(* IEC 61131-3 sources: festo-codesys-mcp/knowledge/library/actuators, 5 files *)

(* ---- FB_ButtonLamp.st ---- *)
(* =============================================================
   FB_ButtonLamp — Illuminated Pushbutton Controller

   Category:     Actuators
   Platform:     CODESYS V3.5 (IEC 61131-3)
   Version:      1.0
   Dependencies: None (standard IEC only)

   Controls an illuminated pushbutton with multiple lamp modes:
   - OFF: Lamp off
   - ON: Lamp solid on
   - BLINK_SLOW: 1Hz blink (500ms on / 500ms off)
   - BLINK_FAST: 4Hz blink (125ms on / 125ms off)

   Also provides edge detection on the button input.

   Usage:
     fbStart : FB_ButtonLamp;
     fbStart(bButton := bDI_StartBtn, nLampMode := 1);
     bStartPressed := fbStart.bPressed;
     bStartLamp    := fbStart.bLamp;
   ============================================================= *)
FUNCTION_BLOCK FB_ButtonLamp
VAR_INPUT
    bButton     : BOOL;                (* Button input (NO contact) *)
    nLampMode   : INT := 0;            (* 0=OFF, 1=ON, 2=BLINK_SLOW, 3=BLINK_FAST *)
END_VAR
VAR_OUTPUT
    bLamp       : BOOL;                (* Lamp output *)
    bPressed    : BOOL;                (* Button is pressed (debounced) *)
    bRising     : BOOL;                (* Rising edge on button *)
    bFalling    : BOOL;                (* Falling edge on button *)
END_VAR
VAR
    tonDebounce : TON;
    rtrigBtn    : R_TRIG;
    ftrigBtn    : F_TRIG;
    tonBlinkOn  : TON;
    tonBlinkOff : TON;
    bBlinkState : BOOL;
    tOnTime     : TIME;
    tOffTime    : TIME;
END_VAR

(* Debounce button *)
tonDebounce(IN := bButton, PT := T#30MS);
bPressed := tonDebounce.Q;

(* Edge detection *)
rtrigBtn(CLK := bPressed);
ftrigBtn(CLK := bPressed);
bRising := rtrigBtn.Q;
bFalling := ftrigBtn.Q;

(* Lamp control *)
CASE nLampMode OF
0: (* OFF *)
    bLamp := FALSE;

1: (* Solid ON *)
    bLamp := TRUE;

2: (* Blink slow — 1Hz *)
    tOnTime := T#500MS;
    tOffTime := T#500MS;
    IF NOT bBlinkState THEN
        tonBlinkOff(IN := TRUE, PT := tOffTime);
        IF tonBlinkOff.Q THEN
            bBlinkState := TRUE;
            tonBlinkOff(IN := FALSE, PT := tOffTime);
        END_IF
    ELSE
        tonBlinkOn(IN := TRUE, PT := tOnTime);
        IF tonBlinkOn.Q THEN
            bBlinkState := FALSE;
            tonBlinkOn(IN := FALSE, PT := tOnTime);
        END_IF
    END_IF
    bLamp := bBlinkState;

3: (* Blink fast — 4Hz *)
    tOnTime := T#125MS;
    tOffTime := T#125MS;
    IF NOT bBlinkState THEN
        tonBlinkOff(IN := TRUE, PT := tOffTime);
        IF tonBlinkOff.Q THEN
            bBlinkState := TRUE;
            tonBlinkOff(IN := FALSE, PT := tOffTime);
        END_IF
    ELSE
        tonBlinkOn(IN := TRUE, PT := tOnTime);
        IF tonBlinkOn.Q THEN
            bBlinkState := FALSE;
            tonBlinkOn(IN := FALSE, PT := tOnTime);
        END_IF
    END_IF
    bLamp := bBlinkState;

ELSE
    bLamp := FALSE;
END_CASE

END_FUNCTION_BLOCK

(* ---- FB_PneumaticCylinder.st ---- *)
(* =============================================================
   FB_PneumaticCylinder — Pneumatic Cylinder Controller

   Category:     Actuators
   Platform:     CODESYS V3.5 (IEC 61131-3)
   Version:      1.0
   Dependencies: None (standard IEC only)

   Controls single-acting or double-acting pneumatic cylinders
   with optional limit switch feedback and timeout monitoring.

   Features:
   - Extend/retract commands with edge detection
   - Limit switch monitoring (extended/retracted sensors)
   - Configurable timeout for fault detection
   - Manual/auto mode support

   Usage:
     fbClamp : FB_PneumaticCylinder;
     fbClamp(bExtend := bCmdClamp, bRetract := bCmdUnclamp,
             bSnsExtended := bDI_ClampFwd, bSnsRetracted := bDI_ClampRev,
             tTimeout := T#3S);
     bClamped   := fbClamp.bExtended;
     bUnclamped := fbClamp.bRetracted;
     bFault     := fbClamp.bErr;
   ============================================================= *)
FUNCTION_BLOCK FB_PneumaticCylinder
VAR_INPUT
    bExtend         : BOOL;                (* Command: extend cylinder *)
    bRetract        : BOOL;                (* Command: retract cylinder *)
    bSnsExtended    : BOOL;                (* Sensor: fully extended *)
    bSnsRetracted   : BOOL;                (* Sensor: fully retracted *)
    tTimeout        : TIME := T#5S;        (* Motion timeout *)
    bDoubleActing   : BOOL := TRUE;        (* TRUE=double-acting, FALSE=spring-return *)
    bEnable         : BOOL := TRUE;        (* Enable control *)
    bReset          : BOOL;                (* Reset error *)
END_VAR
VAR_OUTPUT
    bSolExtend      : BOOL;                (* Solenoid: extend valve *)
    bSolRetract     : BOOL;                (* Solenoid: retract valve (double-acting only) *)
    bExtended       : BOOL;                (* Status: fully extended *)
    bRetracted      : BOOL;                (* Status: fully retracted *)
    bMoving         : BOOL;                (* Status: in motion *)
    bErr          : BOOL;                (* Error: timeout or sensor conflict *)
    nErrId          : DINT;                 (* 0=OK, 1=Extend timeout, 2=Retract timeout, 3=Sensor conflict *)
END_VAR
VAR
    nState          : INT := 0;            (* 0=Idle, 1=Extending, 2=Extended, 3=Retracting, 4=Retracted, 10=Error *)
    tonTimeout      : TON;
    rtrigExtend     : R_TRIG;
    rtrigRetract    : R_TRIG;
END_VAR

rtrigExtend(CLK := bExtend);
rtrigRetract(CLK := bRetract);

(* Sensor conflict detection *)
IF bSnsExtended AND bSnsRetracted THEN
    nState := 10;
    nErrId := 3;
    bErr := TRUE;
    bSolExtend := FALSE;
    bSolRetract := FALSE;
END_IF

(* Reset *)
IF bReset AND bErr THEN
    nState := 0;
    bErr := FALSE;
    nErrId := 0;
    tonTimeout(IN := FALSE, PT := tTimeout);
END_IF

IF NOT bEnable THEN
    bSolExtend := FALSE;
    bSolRetract := FALSE;
    bMoving := FALSE;
    RETURN;
END_IF

CASE nState OF
0: (* Idle *)
    bSolExtend := FALSE;
    bSolRetract := FALSE;
    bMoving := FALSE;
    bExtended := bSnsExtended;
    bRetracted := bSnsRetracted;

    IF rtrigExtend.Q AND NOT bSnsExtended THEN
        nState := 1;
    ELSIF rtrigRetract.Q AND NOT bSnsRetracted THEN
        nState := 3;
    END_IF

1: (* Extending *)
    bSolExtend := TRUE;
    IF bDoubleActing THEN bSolRetract := FALSE; END_IF
    bMoving := TRUE;
    tonTimeout(IN := TRUE, PT := tTimeout);

    IF bSnsExtended THEN
        nState := 2;
        tonTimeout(IN := FALSE, PT := tTimeout);
    ELSIF tonTimeout.Q THEN
        nState := 10;
        nErrId := 1;
        bErr := TRUE;
        bSolExtend := FALSE;
    END_IF

2: (* Extended — hold position *)
    bSolExtend := TRUE;
    IF bDoubleActing THEN bSolRetract := FALSE; END_IF
    bMoving := FALSE;
    bExtended := TRUE;
    bRetracted := FALSE;

    IF rtrigRetract.Q THEN
        nState := 3;
    END_IF

3: (* Retracting *)
    bSolExtend := FALSE;
    IF bDoubleActing THEN bSolRetract := TRUE; END_IF
    bMoving := TRUE;
    tonTimeout(IN := TRUE, PT := tTimeout);

    IF bSnsRetracted THEN
        nState := 4;
        tonTimeout(IN := FALSE, PT := tTimeout);
    ELSIF tonTimeout.Q THEN
        nState := 10;
        nErrId := 2;
        bErr := TRUE;
        IF bDoubleActing THEN bSolRetract := FALSE; END_IF
    END_IF

4: (* Retracted — hold position *)
    bSolExtend := FALSE;
    IF bDoubleActing THEN bSolRetract := FALSE; END_IF
    bMoving := FALSE;
    bExtended := FALSE;
    bRetracted := TRUE;

    IF rtrigExtend.Q THEN
        nState := 1;
    END_IF

10: (* Error *)
    bSolExtend := FALSE;
    bSolRetract := FALSE;
    bMoving := FALSE;

END_CASE

END_FUNCTION_BLOCK

(* ---- FB_PumpManager.st ---- *)
(* =============================================================
   FB_PumpManager — Dual Pump Coordination with Failover

   Category:     Actuators
   Platform:     CODESYS V3.5 (IEC 61131-3)
   Version:      1.0
   Dependencies: None (standard IEC only)

   Manages two pumps with automatic failover, runtime
   equalization, and maintenance hour tracking. Alternates
   primary pump based on accumulated runtime.

   Usage:
     fbPumps : FB_PumpManager;
     fbPumps(
       bEnable   := bCoolingEnable,
       bFlowOK   := bFlowSwitch,
       bPump1OK  := NOT bPump1Fault,
       bPump2OK  := NOT bPump2Fault
     );
     bPump1 := fbPumps.bPump1;
     bPump2 := fbPumps.bPump2;
   ============================================================= *)
FUNCTION_BLOCK FB_PumpManager
VAR_INPUT
    bEnable             : BOOL;             (* Enable pump system *)
    bFlowOK             : BOOL;             (* Flow sensor feedback *)
    bPump1OK            : BOOL := TRUE;     (* Pump 1 healthy *)
    bPump2OK            : BOOL := TRUE;     (* Pump 2 healthy *)
    bSwapPumps          : BOOL;             (* Manual swap command *)
    tFlowCheckDelay     : TIME := T#5S;     (* Delay before flow check *)
    nHoursToSwap        : DINT := 100;      (* Runtime hours before auto-swap *)
END_VAR
VAR_OUTPUT
    bPump1              : BOOL;             (* Pump 1 output *)
    bPump2              : BOOL;             (* Pump 2 output *)
    bFlowAlarm          : BOOL;             (* No flow detected *)
    bBothFaulted        : BOOL;             (* Both pumps faulted *)
    bPumpActive         : BOOL;             (* A pump is running *)
    nActivePump         : INT;              (* 1 or 2 *)
    nRunHours1         : DINT;             (* Pump 1 runtime hours *)
    nRunHours2         : DINT;             (* Pump 2 runtime hours *)
END_VAR
VAR
    bPrimaryIs1         : BOOL := TRUE;     (* TRUE=pump1 is primary *)
    tonFlowCheck        : TON;              (* Flow check delay *)
    tonHourCounter1     : TON;              (* 1-hour timer pump 1 *)
    tonHourCounter2     : TON;              (* 1-hour timer pump 2 *)
    rtrigSwap           : R_TRIG;           (* Swap edge detect *)
    bFailover           : BOOL;             (* Failover active *)
END_VAR

(* ============================================================
   SWAP LOGIC — equalize runtime
   ============================================================ *)

rtrigSwap(CLK := bSwapPumps);

(* Manual swap *)
IF rtrigSwap.Q THEN
    bPrimaryIs1 := NOT bPrimaryIs1;
END_IF;

(* Auto-swap based on runtime hours *)
IF bPrimaryIs1 AND (nRunHours1 - nRunHours2 >= nHoursToSwap) THEN
    bPrimaryIs1 := FALSE;
ELSIF NOT bPrimaryIs1 AND (nRunHours2 - nRunHours1 >= nHoursToSwap) THEN
    bPrimaryIs1 := TRUE;
END_IF;

(* ============================================================
   PUMP SELECTION AND FAILOVER
   ============================================================ *)

IF bEnable THEN
    bBothFaulted := NOT bPump1OK AND NOT bPump2OK;

    IF bBothFaulted THEN
        bPump1 := FALSE;
        bPump2 := FALSE;
        nActivePump := 0;
    ELSIF bPrimaryIs1 THEN
        IF bPump1OK AND NOT bFailover THEN
            bPump1 := TRUE;
            bPump2 := FALSE;
            nActivePump := 1;
        ELSIF bPump2OK THEN
            bPump1 := FALSE;
            bPump2 := TRUE;
            nActivePump := 2;
            bFailover := TRUE;
        ELSE
            bPump1 := TRUE;
            bPump2 := FALSE;
            nActivePump := 1;
        END_IF;
    ELSE
        IF bPump2OK AND NOT bFailover THEN
            bPump1 := FALSE;
            bPump2 := TRUE;
            nActivePump := 2;
        ELSIF bPump1OK THEN
            bPump1 := TRUE;
            bPump2 := FALSE;
            nActivePump := 1;
            bFailover := TRUE;
        ELSE
            bPump1 := FALSE;
            bPump2 := TRUE;
            nActivePump := 2;
        END_IF;
    END_IF;
ELSE
    bPump1 := FALSE;
    bPump2 := FALSE;
    nActivePump := 0;
    bFailover := FALSE;
END_IF;

bPumpActive := bPump1 OR bPump2;

(* ============================================================
   FLOW MONITORING
   ============================================================ *)

tonFlowCheck(IN := bPumpActive, PT := tFlowCheckDelay);
bFlowAlarm := tonFlowCheck.Q AND NOT bFlowOK;

(* On flow alarm, trigger failover *)
IF bFlowAlarm AND NOT bFailover THEN
    bFailover := TRUE;
END_IF;

(* Reset failover when manually swapped or fault clears *)
IF rtrigSwap.Q THEN
    bFailover := FALSE;
END_IF;

(* ============================================================
   RUNTIME HOUR COUNTERS
   ============================================================ *)

tonHourCounter1(IN := bPump1, PT := T#1H);
IF tonHourCounter1.Q THEN
    nRunHours1 := nRunHours1 + 1;
    tonHourCounter1(IN := FALSE);
END_IF;

tonHourCounter2(IN := bPump2, PT := T#1H);
IF tonHourCounter2.Q THEN
    nRunHours2 := nRunHours2 + 1;
    tonHourCounter2(IN := FALSE);
END_IF;

END_FUNCTION_BLOCK

(* ---- FB_SolenoidValve.st ---- *)
(* =============================================================
   FB_SolenoidValve — Solenoid Valve Controller

   Category:     Actuators
   Platform:     CODESYS V3.5 (IEC 61131-3)
   Version:      1.0
   Dependencies: None (standard IEC only)

   Controls a normally-closed or normally-open solenoid valve
   with optional position feedback sensor and stuck-valve detection.

   Usage:
     fbValve : FB_SolenoidValve;
     fbValve(bOpen := bCmdOpenValve, bFeedback := bDI_ValveOpen,
             tFeedbackDelay := T#2S);
     bValveIsOpen := fbValve.bIsOpen;
   ============================================================= *)
FUNCTION_BLOCK FB_SolenoidValve
VAR_INPUT
    bOpen           : BOOL;                (* Command: open valve *)
    bFeedback       : BOOL;                (* Feedback sensor: valve open *)
    bUseFeedback    : BOOL := FALSE;       (* Enable feedback monitoring *)
    tFeedbackDelay  : TIME := T#2S;        (* Feedback timeout *)
    bNormallyOpen   : BOOL := FALSE;       (* TRUE=NO valve, FALSE=NC valve *)
    bEnable         : BOOL := TRUE;        (* Enable control *)
    bReset          : BOOL;                (* Reset error *)
END_VAR
VAR_OUTPUT
    bSolenoid       : BOOL;                (* Solenoid output *)
    bIsOpen         : BOOL;                (* Valve is open *)
    bIsClosed       : BOOL;                (* Valve is closed *)
    bErr          : BOOL;                (* Stuck valve error *)
    nErrId          : DINT;                 (* 0=OK, 1=Stuck open, 2=Stuck closed *)
END_VAR
VAR
    tonFeedback     : TON;
    bExpectedState  : BOOL;
END_VAR

IF bReset THEN
    bErr := FALSE;
    nErrId := 0;
    tonFeedback(IN := FALSE, PT := tFeedbackDelay);
END_IF

IF NOT bEnable THEN
    bSolenoid := bNormallyOpen;  (* De-energize = safe state *)
    bIsOpen := bNormallyOpen;
    bIsClosed := NOT bNormallyOpen;
    RETURN;
END_IF

(* Drive solenoid *)
IF bNormallyOpen THEN
    bSolenoid := NOT bOpen;  (* Energize to close *)
ELSE
    bSolenoid := bOpen;      (* Energize to open *)
END_IF

(* Status *)
IF bUseFeedback THEN
    bIsOpen := bFeedback;
    bIsClosed := NOT bFeedback;

    (* Stuck detection *)
    bExpectedState := bOpen;
    IF bFeedback <> bExpectedState THEN
        tonFeedback(IN := TRUE, PT := tFeedbackDelay);
        IF tonFeedback.Q AND NOT bErr THEN
            bErr := TRUE;
            IF bOpen AND NOT bFeedback THEN
                nErrId := 2; (* Stuck closed *)
            ELSE
                nErrId := 1; (* Stuck open *)
            END_IF
        END_IF
    ELSE
        tonFeedback(IN := FALSE, PT := tFeedbackDelay);
    END_IF
ELSE
    bIsOpen := bOpen;
    bIsClosed := NOT bOpen;
END_IF

END_FUNCTION_BLOCK

(* ---- FB_TankHeater.st ---- *)
(* =============================================================
   FB_TankHeater — Tank Heater with Thermostat and Freeze Protection

   Category:     Actuators
   Platform:     CODESYS V3.5 (IEC 61131-3)
   Version:      1.0
   Dependencies: None (standard IEC only)

   Controls a heating element with thermostat logic (hysteresis),
   overheat protection, freeze protection, dry-run prevention,
   and maximum continuous runtime limit.

   Usage:
     fbHeater : FB_TankHeater;
     fbHeater(
       bEnable   := TRUE,
       bTurnOn   := bCmdHeat,
       rActTemp  := rTankTemperature,
       rSetpoint := 25.0,
       bLevelOK  := bLevelSwitch
     );
     bHeater    := fbHeater.bHeaterElement;
     bTempOK    := fbHeater.bTemperatureOK;
   ============================================================= *)
FUNCTION_BLOCK FB_TankHeater
VAR_INPUT
    bEnable             : BOOL;             (* Enable heater system *)
    bTurnOn             : BOOL;             (* Command to heat *)
    (* Temperature feedback *)
    rActTemp            : REAL;             (* Actual tank temperature [deg C] *)
    rSetpoint           : REAL := 25.0;     (* Target temperature [deg C] *)
    (* Thermostat parameters *)
    rHysteresis         : REAL := 2.0;      (* Hysteresis band [deg C] *)
    rMaxTemp            : REAL := 40.0;     (* Max allowed temperature [deg C] *)
    rMinTemp            : REAL := 5.0;      (* Freeze protection threshold [deg C] *)
    (* Safety *)
    bLevelOK            : BOOL := TRUE;     (* Tank level OK — prevent dry running *)
    tMaxOnTime          : TIME := T#30M;    (* Max continuous heater ON time *)
END_VAR
VAR_OUTPUT
    bHeaterElement      : BOOL;             (* Heater output *)
    bHeating            : BOOL;             (* Heating in progress *)
    bTemperatureOK      : BOOL;             (* Temperature within range *)
    bOverheatAlarm      : BOOL;             (* Over-temperature alarm *)
    bFreezeAlarm        : BOOL;             (* Under-temperature alarm *)
    bTimeoutAlarm       : BOOL;             (* Max ON time exceeded *)
END_VAR
VAR
    bThermostatReq      : BOOL;             (* Internal thermostat state *)
    tonMaxTime          : TON;              (* Max ON timer *)
    tonOverheat         : TON;              (* Overheat confirmation *)
END_VAR

IF NOT bEnable THEN
    bHeaterElement := FALSE;
    bHeating := FALSE;
    bTemperatureOK := TRUE;
    bOverheatAlarm := FALSE;
    bFreezeAlarm := FALSE;
    bTimeoutAlarm := FALSE;
    RETURN;
END_IF;

(* ============================================================
   THERMOSTAT LOGIC WITH HYSTERESIS
   ============================================================ *)

(* Turn ON below setpoint - hysteresis *)
IF rActTemp < (rSetpoint - rHysteresis) THEN
    bThermostatReq := TRUE;
END_IF;

(* Turn OFF above setpoint + hysteresis *)
IF rActTemp > (rSetpoint + rHysteresis) THEN
    bThermostatReq := FALSE;
END_IF;

(* ============================================================
   SAFETY CHECKS
   ============================================================ *)

(* Overheat detection — confirmed after 5s *)
tonOverheat(IN := rActTemp > rMaxTemp, PT := T#5S);
bOverheatAlarm := tonOverheat.Q;

(* Freeze protection — always heat if too cold *)
bFreezeAlarm := rActTemp < rMinTemp;

(* Maximum continuous runtime *)
tonMaxTime(IN := bHeaterElement, PT := tMaxOnTime);
bTimeoutAlarm := tonMaxTime.Q;

(* ============================================================
   OUTPUT LOGIC
   ============================================================ *)

(* Heater ON conditions:
   1. Enabled AND commanded on (or freeze protection)
   2. Thermostat requests heat (or freeze protection)
   3. Water level OK (prevent dry-run)
   4. No overheat
   5. Max time not exceeded *)
bHeaterElement := bEnable AND
                  (bTurnOn OR bFreezeAlarm) AND
                  (bThermostatReq OR bFreezeAlarm) AND
                  bLevelOK AND
                  NOT bOverheatAlarm AND
                  NOT bTimeoutAlarm;

bHeating := bHeaterElement;

(* Temperature status *)
bTemperatureOK := (rActTemp >= rMinTemp) AND (rActTemp <= rMaxTemp);

END_FUNCTION_BLOCK
